PROGRAM Printing
VAR
	CadModel: BOOL;
	StlFile: BOOL;
	Preheat: BOOL;
	EntrySlice: BOOL;
	PrintSettings: BOOL;
	Slice: BOOL;
	TransferFile: BOOL;
	PreheatTimer :TON;
	EntryPrint: BOOL;
	StartPrint: BOOL;
	Checkprint1: BOOL;
	ContinuePrint: BOOL;
	PrintComplete: BOOL;
	FinishPrintEntry: BOOL;
	RemovePrint: BOOL;
	CleanBed: BOOL;
	PrintSucceeded: BOOL;
	PrintFinished: BOOL;
	PrintFailed:BOOL;
	PrintStatePrepareModel: BOOL;
	PrintStateSlicePrint: BOOL;
	PrintStatePrint: BOOL;
	PrintStateFinishPrint: BOOL;
END_VAR


CASE gvl.PrintState OF

//Prepare state for modeling and converting 3d-print	
PrintingStates.PrepareModel:
PrintStatePrepareModel:=TRUE;
PrintStateSlicePrint:=FALSE;
PrintStatePrint:=FALSE;
PrintStateFinishPrint:=FALSE;

IF gvl.EntryPrint = TRUE THEN
	gvl.EntryPrint := FALSE;
	CadModel := TRUE;
END_IF
IF Cadmodel = TRUE THEN
	StlFile :=TRUE;
	Cadmodel:=FALSE;
END_IF
IF StlFile = TRUE THEN
	Preheat :=TRUE;
	StlFile:=FALSE;
END_IF
IF Preheat = TRUE THEN
	gvl.PrintState := printingstates.SlicePrint;
	Preheat := FALSE;
	EntrySlice :=TRUE;
END_IF

//Second State, Slice the print
PrintingStates.SlicePrint:
PrintStatePrepareModel:=FALSE;
PrintStateSlicePrint:=TRUE;
PrintStatePrint:=FALSE;
PrintStateFinishPrint:=FALSE;

PreheatTimer(in:=TRUE,PT:=T#10S); //preheat printer
IF EntrySlice = TRUE THEN
	EntrySlice:=FALSE;
	PrintSettings:=TRUE;	
END_IF
IF PrintSettings THEN
	PrintSettings:= FALSE;
	Slice :=TRUE;
END_IF
IF Slice THEN
	Slice :=FALSE;
	TransferFile:=TRUE;
END_IF
IF Transferfile = TRUE AND PreheatTimer.Q = TRUE THEN
	TransferFile:=FALSE;
	GVL.PrintState :=PrintingStates.Print;
	EntryPrint:=TRUE;
END_IF

//Third state of printing
PrintingStates.Print:
PrintStatePrepareModel:=FALSE;
PrintStateSlicePrint:=FALSE;
PrintStatePrint:=TRUE;
PrintStateFinishPrint:=FALSE;

IF EntryPrint THEN
	Entryprint :=FALSE;	
	StartPrint := TRUE;
END_IF
IF Startprint THEN
	Startprint := FALSE;
	Checkprint1 := TRUE;
	gvl.PrintStarted:=TRUE; //Signal to start Running routine
END_IF

IF Checkprint1 THEN 
	IF gvl.Layer1Good = TRUE THEN //If the first layer is good, continue proces and start running proces
		Checkprint1:=FALSE;			//Button in visualization to make true
		ContinuePrint := TRUE;
		
	ELSIF gvl.Layer1Bad = TRUE THEN
	checkprint1 := FALSE;
	GVL.PrintState := printingstates.SlicePrint; //If the first layer failed, go back to the slicing settings	
	END_IF
END_IF
IF ContinuePrint THEN
	ContinuePrint:=FALSE;
	PrintComplete:= TRUE;
END_IF
IF PrintComplete THEN
	GVL.PrintState:=PrintingStates.FinishPrint;
	PrintComplete:=FALSE;
	FinishPrintEntry:=TRUE;
END_IF

//Last state of printing proces
PrintingStates.FinishPrint:
PrintStatePrepareModel:=FALSE;
PrintStateSlicePrint:=FALSE;
PrintStatePrint:=FALSE;
PrintStateFinishPrint:=TRUE;
IF FinishPrintEntry THEN
	FinishPrintEntry:=FALSE;
	RemovePrint:=TRUE;
END_IF
IF Removeprint THEN
	Removeprint:=FALSE;
	CleanBed:=TRUE;
END_IF
IF CleanBed THEN
	IF PrintSucceeded THEN //Button in visualization to make true
		PrintFinished:=TRUE;
		CleanBed:=FALSE;
	ELSIF PrintFailed THEN
		gvl.PrintState:=PrintingStates.SlicePrint;
		CleanBed:=FALSE;
		EntrySlice:= TRUE;
	END_IF
END_IF
IF printFinished THEN
	gvl.PrintFinished:=TRUE;
	PrintFinished:=FALSE;
	gvl.Printstate:=PrintingStates.PrepareModel;
END_IF

END_CASE

END_PROGRAM

(* stored: Version 1.1.0.1, ProductVersion 3.1.4024.15
   POU Printing: Id {5d1dbc66-6bdd-4670-8314-e29a9e50c9f9}, SpecialFunc None *)
